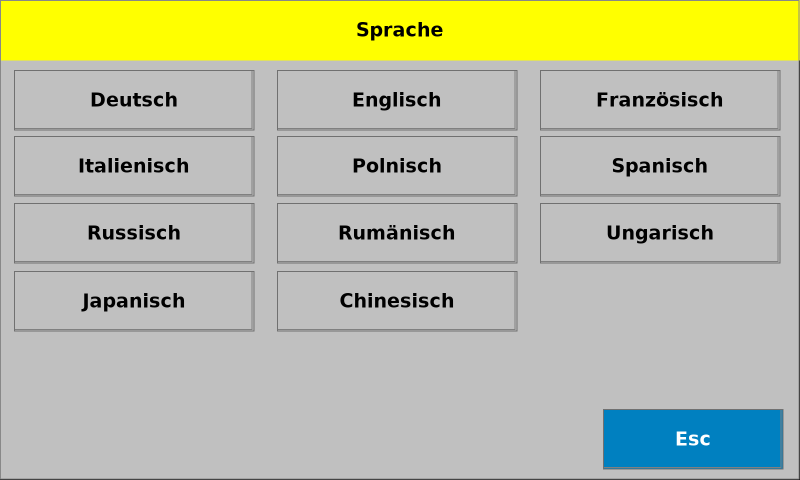
VISUALIZATION Sprache  // 800x480
    Rectangle (0,0 800x480)
    Rectangle (0,0 800x60), "Sprache"
    Button (14,70 240x60), "Deutsch"
        OnMouseUp: ChangeLanguage ChangeLanguage=de
    Button (14,136 240x60), "Italienisch"
        OnMouseUp: ChangeLanguage ChangeLanguage=IT
    Button (14,203 240x60), "Russisch"
        OnMouseUp: ChangeLanguage ChangeLanguage=RU
    Button (277,70 240x60), "Englisch"
        OnMouseUp: ChangeLanguage ChangeLanguage=EN
    Button (277,136 240x60), "Polnisch"
        OnMouseUp: ChangeLanguage ChangeLanguage=PL
    Button (277,203 240x60), "Rumänisch"
        OnMouseUp: ChangeLanguage ChangeLanguage=RO
    Button (603,409 180x60), "Esc"
        OnMouseUp: change screen: Start
        OnMouseUp: execute { P_SaveCurrentLanguage(); }
    Button (540,70 240x60), "Französisch"
        OnMouseUp: ChangeLanguage ChangeLanguage=FR
    Button (540,136 240x60), "Spanisch"
        OnMouseUp: ChangeLanguage ChangeLanguage=ES
    Button (540,203 240x60), "Ungarisch"
        OnMouseUp: ChangeLanguage ChangeLanguage=HU
    Button (14,271 240x60), "Japanisch"
        OnMouseUp: ChangeLanguage ChangeLanguage=JA
    Button (277,271 240x60), "Chinesisch"
        OnMouseUp: ChangeLanguage ChangeLanguage=ZH
END_VISUALIZATION

(* stored: Version 1.1.0.1, ProductVersion 3.1.4024.3
   Visu Sprache: Id {496cd653-7d8c-49bd-ae86-897da963f0ac} *)
